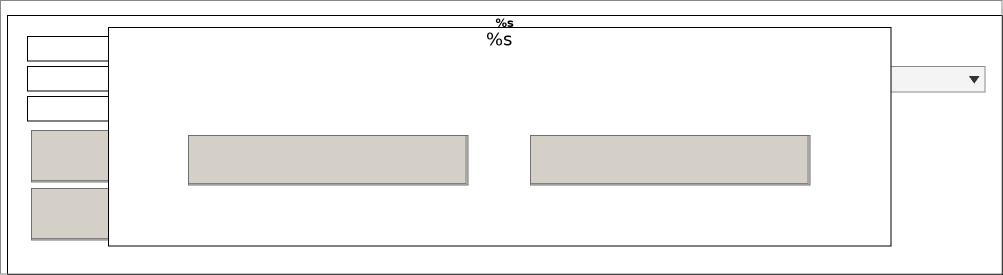
VISUALIZATION VISU_PARAMETRAGE_RELAY  // 1003x275
VAR_IN_OUT
	COM : BLOCK_RS232_ONBOARD_V4;
END_VAR
    RoundedRectangle (7,15 996x260), "%s", text list: 'TextList_CryoPump', text index: 80
    Rectangle (27,36 475x25), text list: 'TextList_CryoPump', text index: 66
    Rectangle (502,36 349x25), "%i", text variable: COM.PRM_Relay, input disabled if: NOT Global_Variables.PRG_USER.ACTU_USER.CONF_MACHINE
        OnMouseClick: write COM.PRM_Relay via Edit, min 1, max 2
    Rectangle (27,66 475x25), text list: 'TextList_CryoPump', text index: 67
    Rectangle (27,96 475x25), invisible if: COM.VAR_Visibilite_valeur_relay, text list: 'TextList_CryoPump', text index: 68
    Rectangle (502,96 349x25), "%i", text variable: COM.PRM_Valeur, invisible if: COM.VAR_Visibilite_valeur_relay, input disabled if: NOT Global_Variables.PRG_USER.ACTU_USER.CONF_MACHINE
        OnMouseClick: write COM.PRM_Valeur via Edit
    Button (31,130 244x52), input disabled if: NOT Global_Variables.PRG_USER.ACTU_USER.CONF_MACHINE, text list: 'TextList_CryoPump', text index: 69
        OnMouseDown: execute { COM.Message_alerte_invisible:=false; }
    Rectangle (485,158 200x26), text list: 'TextList_CryoPump', text index: COM.VAR_Affichage_Commande_Relay
    Rectangle (685,158 200x26), "%s", text variable: COM.VAR_Affichage_Valeur_Relay
    Rectangle (685,133 200x26), "mode", text list: 'TextList_CryoPump', text index: BOOL_TO_INT(COM.TAB_Affichage_Mode_relay[COM.PRM_Relay])+81
    Rectangle (485,184 200x26), "delay", text list: 'TextList_CryoPump', text index: 74
    Rectangle (685,184 200x26), "%s sec", text variable: COM.VAR_Affichage_ValeurTIME_Relay
    Button (31,188 244x52), input disabled if: NOT Global_Variables.PRG_USER.ACTU_USER.CONF_MACHINE, text list: 'TextList_CryoPump', text index: 85
        OnMouseDown: execute { COM.Message_alerte_invisible:=false; }
    ComboBoxInteger (503,66 482x26), variable: COM.PRM_Action, input disabled if: NOT Global_Variables.PRG_USER.ACTU_USER.CONF_MACHINE, text list: 'TextList_Cryo_Relays_Parameters'
    Button (281,130 198x52), text list: 'TextList_CryoPump', text index: 88
        OnMouseDown: execute { COM.CO_Lecture_Relay:=TRUE; }
        OnMouseUp: execute { COM.CO_Lecture_Relay:=false; }
    Button (281,188 197x52), input disabled if: NOT Global_Variables.PRG_USER.ACTU_USER.CONF_MACHINE, text list: 'TextList_CryoPump', text index: 36
        OnMouseDown: execute { COM.Message_confirm_invisible:=false; }
        OnMouseUp: execute {  }
    Group (109,27 782x218)
        Rectangle (0,0 587x176), "%s", invisible if: COM.Message_alerte_invisible, text list: 'TextList_CryoPump', text index: 89
        Rectangle (6,39 579x68), "%s", invisible if: COM.Message_alerte_invisible, text list: 'TextList_CryoPump', text index: 90
        Button (60,120 213x42), invisible if: COM.Message_alerte_invisible, text list: 'TextList_CryoPump', text index: 92
            OnMouseDown: execute { COM.CO_Envoie_Param_Relay:=true; }
            OnMouseUp: execute { COM.Message_alerte_invisible:=TRUE; }
            OnMouseUp: execute { COM.CO_Envoie_Param_Relay:=false; }
        Button (323,120 211x41), invisible if: COM.Message_alerte_invisible, text list: 'TextList_CryoPump', text index: 93
            OnMouseDown: execute { COM.Message_alerte_invisible:=true; }
    Group (109,28 782x216), invisible if: COM.Message_alerte_invisible2
        Rectangle (0,0 587x176), "%s", invisible if: COM.Message_alerte_invisible, text list: 'TextList_CryoPump', text index: 89
        Rectangle (6,39 579x68), "%s", invisible if: COM.Message_alerte_invisible, text list: 'TextList_CryoPump', text index: 90
        Button (319,120 210x40), invisible if: COM.Message_alerte_invisible, text list: 'TextList_CryoPump', text index: 93
            OnMouseDown: execute { COM.Message_alerte_invisible:=true; }
        Button (63,120 210x40), text list: 'TextList_CryoPump', text index: 85
            OnMouseDown: execute { COM.CO_Envoie_Param_Relay:=true; }
            OnMouseUp: execute { COM.CO_Envoie_Param_Relay:=FALSE; }
            OnMouseUp: execute { COM.PRM_Mode := TRUE; }
    Group (108,27 783x219)
        Rectangle (0,0 783x219), "%s", invisible if: COM.Message_confirm_invisible, text list: 'TextList_CryoPump', text index: 91
        Button (422,108 280x50), invisible if: COM.Message_confirm_invisible, text list: 'TextList_CryoPump', text index: 93
            OnMouseDown: execute { COM.Message_confirm_invisible:=true; }
        Button (80,108 280x50), invisible if: COM.Message_confirm_invisible, text list: 'TextList_CryoPump', text index: 92
            OnMouseDown: execute { COM.CO_Param_usine_Relay:=TRUE; }
            OnMouseUp: execute { COM.CO_Param_usine_Relay:=FALSE; }
            OnMouseUp: execute { COM.Message_confirm_invisible:=true; }
END_VISUALIZATION

(* stored: Version 1.1.0.1, ProductVersion 3.1.4026.18
   Visu VISU_PARAMETRAGE_RELAY: Id {2b035eb2-48e3-423e-b2b4-38724544cdd6} *)
